Universal Robots PolyScope program: 01_Pick_Place_01.urp

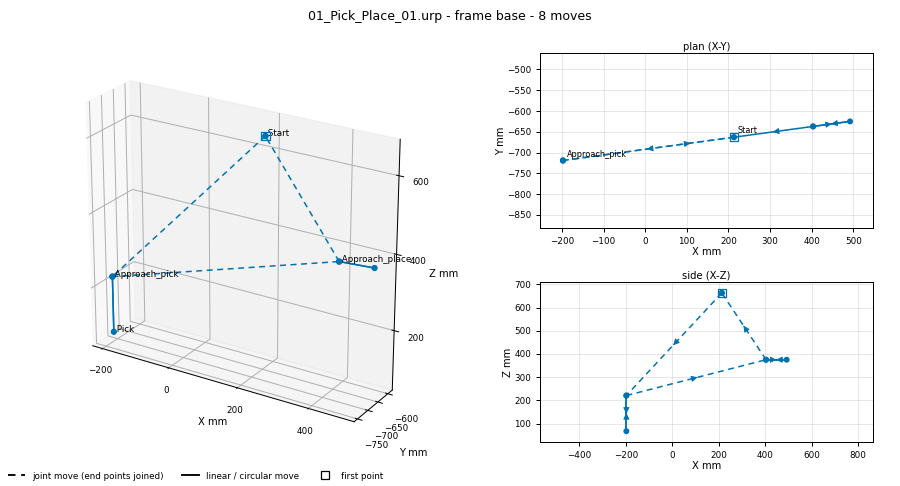
[picture p0: tool path of 01_Pick_Place_01.urp in frame base, 8 of 8 moves have a stored position in this frame; points joined in program order, loops and branches not executed]
Program 01_Pick_Place_01 (installation=default directory=/home/ur/ursim-current/programs/Test_Programs createdIn=5.9.1.1031110 lastSavedIn=5.9.1.1031110 robotSerialNumber=20195599999)
Calibrated DH parameters: a=[0, -0.425, -0.3922, 0, 0, 0]; d=[0.1625, 0, 0, 0.1333, 0.0997, 0.0996]; alpha=[1.570796, 0, 0, 1.570796, -1.570796, 0]; deltaTheta=[0, 0, 0, 0, 0, 0]
Robot Program (runOnlyOnce=false)
  MoveJ speed 60 deg/s, acceleration 80 deg/s^2 (useActiveTCP=true) feature=Base
    Waypoint Start: TCP in base x=213.227 y=-662.982 z=662.763 mm, rx=0 ry=-2.2214 rz=2.2214 rad; joints [97.946, -62.545, 59.12, 183.425, -97.946, -0.001] deg
    Waypoint Approach_pick: TCP in base x=-197.817 y=-718.988 z=221.036 mm, rx=-0.2834 ry=3.1288 rz=0 rad; joints [64.319, -49.221, 73.889, 245.332, -90, -36.031] deg
    MoveL speed 250 mm/s, acceleration 1200 mm/s^2 (useActiveTCP=true) feature=Base
      Waypoint Pick: TCP in base x=-197.817 y=-718.988 z=67.509 mm, rx=-0.2834 ry=3.1288 rz=0 rad; joints [64.319, -37.701, 78.314, 229.387, -90, -36.031] deg
      Wait Sleep waitTime=2
      Waypoint Approach_pick: TCP in base x=-197.817 y=-718.988 z=221.036 mm, rx=-0.2834 ry=3.1288 rz=0 rad; joints [64.319, -49.221, 73.889, 245.332, -90, -36.031] deg
    MoveJ speed 60 deg/s, acceleration 80 deg/s^2 (useActiveTCP=true) feature=Base
      Waypoint Approach_place: TCP in base x=403.469 y=-637.06 z=375.22 mm, rx=-0.1421 ry=1.5693 rz=0.0707 rad; joints [104.411, -37.423, 59.079, 160.559, -6.657, 85.209] deg
    MoveL speed 250 mm/s, acceleration 1200 mm/s^2 (useActiveTCP=true) feature=Base
      Waypoint Place: TCP in base x=492.291 y=-624.958 z=375.22 mm, rx=-0.1421 ry=1.5693 rz=0.0707 rad; joints [111.418, -32.036, 48.623, 164.5, -13.661, 86.353] deg
      Wait Sleep waitTime=2
      Waypoint Approach_place: TCP in base x=403.469 y=-637.06 z=375.22 mm, rx=-0.1421 ry=1.5693 rz=0.0707 rad; joints [104.411, -37.423, 59.079, 160.559, -6.657, 85.209] deg
    MoveJ speed 60 deg/s, acceleration 80 deg/s^2 (useActiveTCP=true) feature=Base
      Waypoint Start: TCP in base x=213.227 y=-662.982 z=662.763 mm, rx=0 ry=-2.2214 rz=2.2214 rad; joints [97.946, -62.545, 59.12, 183.425, -97.946, -0.001] deg
